Fanuc KAREL source: kt00488.KL

-- PROVISIONAL review KL for V1013-1; original PC SHA256 c5611d3ff4f0bf26b6d650b417e9160ff46ff9543de1a34b7f73ec9911248761
-- Incomplete behavior may be omitted. Consult companion uncertainty JSON. Do not deploy.
PROGRAM KT00488
%NOLOCKGROUP
VAR
  OUT : BOOLEAN
-- UNRESOLVED_DECL P1 type=000101
-- UNRESOLVED_DECL P2 type=000199
BEGIN
  -- UNRESOLVED_PC offsets 5-33; opcodes 49,49,7E,AC,23
  -- UNRESOLVED_PC offsets 38-42; opcodes 7F
END KT00488
